FUNCTION ReplaceStep : bool
VAR_INPUT
	step:ST_Tableau;
END_VAR
VAR
END_VAR

//change l'étape actuelle
G_Match.Tableau[G_Match.iLigne] := step;

END_FUNCTION

(* stored: Version 1.1.0.1, ProductVersion 3.1.4024.12
   POU ReplaceStep: Id {a91df4fa-cd8a-488c-8cb8-ec84394d75a6}, SpecialFunc None *)
